INTERFACE I_Extends EXTENDS I_Base

END_INTERFACE

(* stored: Version 1.1.0.1
   Itf I_Extends: Id {44444444-4444-4444-4444-444444444405} *)
